// TwinCAT 3 PLC project Untitled1
// ProgramVersion: 3.1.4024.0
// libraries:
//   Tc2_Standard, * (Beckhoff Automation GmbH)
//   Tc2_System, * (Beckhoff Automation GmbH)
//   Tc3_Module, * (Beckhoff Automation GmbH)
//   VisuSymbols,3.5.10.0,System
// project tree:
//   / GlobalTextList.TcGTLO, Task_1.TcTTO, Task_2.TcTTO
//   GVLs/ GVL_Carbid.TcGVL
//   POUs/ UserTask.TcPOU, BusTask.TcPOU
//   VISUs/ VisualizationManager.TcVMO (not stored), Visualization_Carbid_V2.TcVIS
// real-time tasks:
//   TASK Task_1: cycle T#10ms, priority 1, ADS port 351
//   TASK Task_2: cycle T#10ms, priority 2, ADS port 352

CONFIGURATION Untitled1
    RESOURCE PLC ON TwinCAT3
        TASK Task_1(INTERVAL := T#10ms, PRIORITY := 1);
        TASK Task_2(INTERVAL := T#10ms, PRIORITY := 2);
        PROGRAM UserTask WITH Task_1 : UserTask;
        PROGRAM BusTask WITH Task_2 : BusTask;
    END_RESOURCE
END_CONFIGURATION

// ---- GVLs/GVL_Carbid.TcGVL
VAR_GLOBAL
    (* Var voor testen later verwijderen*)
	Button : BOOL;
	Lamp : BOOL;
	BlinkingLamp : BOOL;

	(* UserTask-variabelen *)
    UserStep : INT := 0;
	StartProcess : BOOL;
    AddCarbid : BOOL;
    AddWater : BOOL;
    PlaceBall : BOOL;
    FlameOn : BOOL;
    Fire : BOOL := FALSE;
	CheckAfterShot : BOOL := FALSE;
	RetrieveBall  : BOOL := FALSE;

    (* BusTask-variabelen *)
    BusStep : INT := 0;
    CarbidAdded : BOOL := FALSE;
	WaterAdded : BOOL := FALSE;
	BallPlaced : BOOL := FALSE;
	GasFormation : BOOL := FALSE;
    EnoughGas : BOOL := FALSE;
    ReadyToFire : BOOL := FALSE;
    RemoveDebris : BOOL := FALSE;
END_VAR

// ---- POUs/UserTask.TcPOU
PROGRAM UserTask
VAR
    tUserDelay : TON;  (* Timer voor gebruikersacties *)
END_VAR

(* Testen of VISU werkt later verwijderen *)
IF GVL_Carbid.Button THEN
   GVL_Carbid.Lamp := TRUE;    (* Zet lamp aan *)
ELSE
   GVL_Carbid.Lamp := FALSE;   (* Zet lamp uit *)
END_IF

(* Proces start door de gebruiker *)
IF GVL_Carbid.StartProcess THEN
    CASE GVL_Carbid.UserStep OF
        0:  (* Voeg carbid toe *)
            GVL_Carbid.AddCarbid := TRUE;
            IF GVL_Carbid.CarbidAdded THEN
                GVL_Carbid.AddCarbid := FALSE;
                GVL_Carbid.UserStep := 1; (* Ga naar de volgende stap *)
            END_IF;

        1:  (* Voeg water toe *)
            GVL_Carbid.AddWater := TRUE;
            IF GVL_Carbid.WaterAdded THEN   (* Communicatie met BusTask *)
                GVL_Carbid.AddWater := FALSE;
                GVL_Carbid.UserStep := 2;
            END_IF;

        2:  (* Plaats bal in bus *)
            GVL_Carbid.PlaceBall := TRUE;
            tUserDelay(IN := TRUE, PT := T#2S); (* Voeg 2 seconden vertraging toe *)
            IF tUserDelay.Q THEN
                GVL_Carbid.PlaceBall := FALSE;
                GVL_Carbid.BallPlaced := TRUE;  (* Communicatie met BusTask *)
                GVL_Carbid.UserStep := 3;
                tUserDelay(IN := FALSE);
            END_IF;

        3:  (* Wacht op vuur *)
            IF GVL_Carbid.BallPlaced AND GVL_Carbid.FlameOn THEN
                GVL_Carbid.Fire := TRUE; (* Vuurt af *)
                GVL_Carbid.UserStep := 4;
            END_IF;

        4:  (* Controleer bus na schot *)
            GVL_Carbid.CheckAfterShot := TRUE;
            tUserDelay(IN := TRUE, PT := T#2S); (* Voeg 2 seconden vertraging toe *)
            IF tUserDelay.Q THEN
                GVL_Carbid.CheckAfterShot := FALSE;
                GVL_Carbid.UserStep := 5;
                tUserDelay(IN := FALSE);
            END_IF;

        5:  (* Haal de bal op *)
            GVL_Carbid.RetrieveBall := TRUE;
            tUserDelay(IN := TRUE, PT := T#2S); (* Voeg 2 seconden vertraging toe *)
            IF tUserDelay.Q THEN
                GVL_Carbid.RetrieveBall := FALSE;
                GVL_Carbid.UserStep := 0;  (* Reset naar begin *)
                tUserDelay(IN := FALSE);
            END_IF;
    END_CASE;
END_IF;

END_PROGRAM

// ---- POUs/BusTask.TcPOU
PROGRAM BusTask
VAR
    tBusDelay : TON;        (* Timer voor busacties *)
    tCarbidReaction : TON;  (* Timer voor gasvorming proces *)
    tBlink : TON;           (* Timer voor knipperen van ReadyToFire *)
    BlinkState : BOOL := FALSE;  (* Knipperstatus voor ReadyToFire *)
END_VAR

(* Testen of VISU werkt later verwijderen *)
IF GVL_Carbid.Lamp THEN
    tBlink(IN := TRUE, PT := T#500MS);
    IF tBlink.Q THEN
        blinkState := NOT blinkState;
        GVL_Carbid.BlinkingLamp := blinkState;  (* Laat lamp knipperen *)
        tBlink(IN := FALSE);  (* Reset de timer *)
    END_IF;
ELSE
    GVL_Carbid.BlinkingLamp := FALSE;  (* Zet lamp uit als GVL_Carbid.Lamp uit is *)
END_IF

(* Beheer processen in de bus *)
CASE GVL_Carbid.BusStep OF
    0:  (* Wacht op carbid toevoeging *)
        IF GVL_Carbid.AddCarbid THEN
			tBusDelay(IN := TRUE, PT := T#2S); (* Voeg 2 seconden vertraging toe *)
			IF tBusDelay.Q THEN
                GVL_Carbid.CarbidAdded := TRUE;
                GVL_Carbid.BusStep := 1; (* Ga naar de volgende stap *)
                tBusDelay(IN := FALSE); (* Reset timer voor volgende stap *)
            END_IF;
        END_IF;

    1:  (* Wacht op water toevoeging *)
        IF GVL_Carbid.AddWater THEN
            tBusDelay(IN := TRUE, PT := T#2S); (* Gasvorming duurt 10 seconden *)
            IF tBusDelay.Q THEN
				GVL_Carbid.WaterAdded := TRUE;
                GVL_Carbid.GasFormation := TRUE;
                GVL_Carbid.BusStep := 2;
                tBusDelay(IN := FALSE);
            END_IF;
        END_IF;
		
	2:	(* Wacht op genoeg gas *)
		IF GVL_Carbid.GasFormation THEN
			tCarbidReaction(IN := TRUE, PT := T#10S); (* Gasvorming duurt 10 seconden *)
            IF tCarbidReaction.Q THEN
                GVL_Carbid.EnoughGas := TRUE;
				GVL_Carbid.GasFormation := FALSE;
                GVL_Carbid.BusStep := 3;
                tCarbidReaction(IN := FALSE);
            END_IF;
		END_IF

    3:  (* Ready to Fire knippert als er genoeg gas is *)
        IF GVL_Carbid.EnoughGas AND GVL_Carbid.BallPlaced THEN
            tBlink(IN := TRUE, PT := T#500MS);  (* Knipperen elke 500 ms *)
            IF tBlink.Q THEN
                blinkState := NOT blinkState;  (* Wissel tussen aan en uit *)
                GVL_Carbid.ReadyToFire := blinkState;
            END_IF;
            (* Ga naar de vuurfase wanneer de gebruiker het aangeeft *)
            IF GVL_Carbid.Fire THEN
                GVL_Carbid.Fire := TRUE;
                GVL_Carbid.BusStep := 4;
            END_IF;
        END_IF;

    4:  (* Vuur de bal af *)
        GVL_Carbid.ReadyToFire := FALSE; (* Stop Ready to Fire *)
		GVL_Carbid.WaterAdded := FALSE;
		GVL_Carbid.CarbidAdded := FALSE;
		GVL_Carbid.EnoughGas := FALSE;
		GVL_Carbid.BallPlaced := FALSE;
        GVL_Carbid.Fire := TRUE;  (* Afvuren *)
        GVL_Carbid.BusStep := 5;

    5:  (* Reset het systeem na het schot *)
        GVL_Carbid.Fire := FALSE;
        GVL_Carbid.RemoveDebris := TRUE;
        tBusDelay(IN := TRUE, PT := T#2S);  (* 2 seconden voor opruimen *)
        IF tBusDelay.Q THEN
            GVL_Carbid.RemoveDebris := FALSE;
            GVL_Carbid.BusStep := 0;  (* Reset bus *)
            tBusDelay(IN := FALSE);
        END_IF;
END_CASE;

END_PROGRAM

// ---- GlobalTextList.TcGTLO
TEXTLIST GlobalTextList
  985 = 'AddCarbid'
  878 = 'AddWater'
  597 = 'BallPlaced'
  49 = 'BallSealed'
  69 = 'Bus_Visu'
  500 = 'CarbidAdded'
  387 = 'CheckAfterShot'
  882 = 'EnoughGas'
  914 = 'EnoughWater'
  48 = 'Fire'
  896 = 'FlameOn'
  578 = 'GasFormation'
  201 = 'Mis leuk om de hoeveelheid water te zien oplopen en dan als het gas vormt zie je het weer omlaag gaan tot alle gas gevormd is'
  395 = 'PlaceBall'
  935 = 'ReadyToFire'
  771 = 'RemoveDebris'
  117 = 'RetrieveBall'
  750 = 'RetriveBall'
  450 = 'StartProcess'
  129 = 'TEST VISU'
  333 = 'User_Visu'
  341 = 'WaterAdded'
END_TEXTLIST

// ---- VISUs/Visualization_Carbid_V2.TcVIS
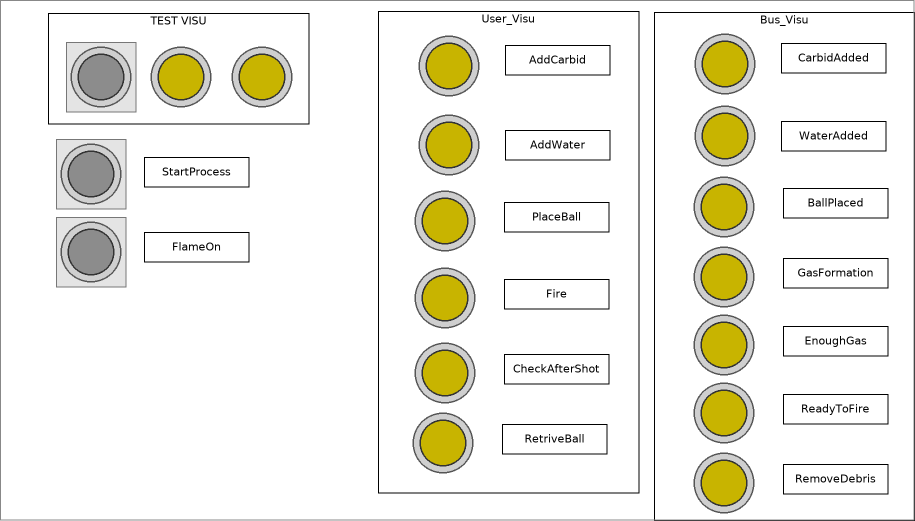
VISUALIZATION Visualization_Carbid_V2  // 915x521
    Rectangle (378,11 261x482), "User_Visu"
    Rectangle (48,13 261x111), "TEST VISU"
    Lamp1 (146,42 70x70), variable: Lamp, style: Lamp-Lamp1-Yellow
    PushSwitch (66,42 70x70), variable: Button, behaviour: TAP, style: Switch-PushSwitch-Gray
    Lamp1 (227,42 70x70), variable: BlinkingLamp, style: Lamp-Lamp1-Yellow
    PushSwitchLed (56,139 70x70), variable: StartProcess, behaviour: TOGGLE, style: Switch-PushSwitchLed-Gray
    PushSwitch (56,217 70x70), variable: FlameOn, behaviour: TAP, style: Switch-PushSwitch-Gray
    Rectangle (144,157 105x30), "StartProcess"
    Rectangle (144,232 105x30), "FlameOn"
    Lamp1 (414,31 70x70), variable: AddCarbid, style: Lamp-Lamp1-Yellow
    Lamp1 (414,110 70x70), variable: AddWater, style: Lamp-Lamp1-Yellow
    Rectangle (505,45 105x30), "AddCarbid"
    Rectangle (505,130 105x30), "AddWater"
    Lamp1 (410,186 70x70), variable: PlaceBall, style: Lamp-Lamp1-Yellow
    Rectangle (504,202 105x30), "PlaceBall"
    Lamp1 (410,263 70x70), variable: Fire, style: Lamp-Lamp1-Yellow
    Rectangle (504,279 105x30), "Fire"
    Lamp1 (410,338 70x70), variable: CheckAfterShot, style: Lamp-Lamp1-Yellow
    Rectangle (504,354 105x30), "CheckAfterShot"
    Rectangle (654,12 261x509), "Bus_Visu"
    Lamp1 (690,29 70x70), variable: CarbidAdded, style: Lamp-Lamp1-Yellow
    Lamp1 (690,101 70x70), variable: WaterAdded, style: Lamp-Lamp1-Yellow
    Rectangle (781,43 105x30), "CarbidAdded"
    Rectangle (781,121 105x30), "WaterAdded"
    Lamp1 (689,242 70x70), variable: GasFormation, style: Lamp-Lamp1-Yellow
    Rectangle (783,258 105x30), "GasFormation"
    Lamp1 (689,310 70x70), variable: EnoughGas, style: Lamp-Lamp1-Yellow
    Rectangle (783,326 105x30), "EnoughGas"
    Lamp1 (689,378 70x70), variable: ReadyToFire, style: Lamp-Lamp1-Yellow
    Rectangle (783,394 105x30), "ReadyToFire"
    Lamp1 (408,408 70x70), variable: RetrieveBall, style: Lamp-Lamp1-Yellow
    Rectangle (502,424 105x30), "RetriveBall"
    Lamp1 (689,448 70x70), variable: RemoveDebris, style: Lamp-Lamp1-Yellow
    Rectangle (783,464 105x30), "RemoveDebris"
    Lamp1 (689,172 70x70), variable: BallPlaced, style: Lamp-Lamp1-Yellow
    Rectangle (783,188 105x30), "BallPlaced"
END_VISUALIZATION
